(* PLC project add_syrup, Dassault Systèmes ControlBuild 2024x *)
(* stored: creationDateTime 2023-10-03T11:13:37-01:00 *)

FUNCTION_BLOCK batch.add_syrup
  VAR_INPUT
    flowSyrup1 : REAL := 0.0;
    flowSyrup2 : REAL := 0.0;
    flowSyrup3 : REAL := 0.0;
  END_VAR
  VAR_OUTPUT
    flow : REAL := 0.0;
  END_VAR

IF (flowSyrup1+flowSyrup2+flowSyrup3>0.0) THEN
	flow := flowSyrup1+flowSyrup2+flowSyrup3;
ELSE
	flow := 0.0;
END_IF;
END_FUNCTION_BLOCK
